FUNCTION_BLOCK PY_RELAY_CTRL (* Basic FB with empty ECC *)
  {SET_ATTRIBUTE(OpcUa, SERVICE)}
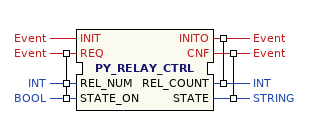
  EVENT_INPUT
    INIT;
    REQ WITH REL_NUM, STATE_ON;
  END_EVENT
  EVENT_OUTPUT
    INITO WITH REL_COUNT;
    CNF WITH STATE;
  END_EVENT
  VAR_INPUT
    REL_NUM : INT; {SET_ATTRIBUTE(OpcUa, Variable.REQ)}
    STATE_ON : BOOL; {SET_ATTRIBUTE(OpcUa, Variable.REQ)}
  END_VAR
  VAR_OUTPUT
    REL_COUNT : INT; {SET_ATTRIBUTE(OpcUa, Variable.INIT)}
    STATE : STRING; {SET_ATTRIBUTE(OpcUa, Variable.REQ)}
  END_VAR
END_FUNCTION_BLOCK
